RoboDK station: Double suction HAMK Robotics station MG400 Wood Sticks.rdk

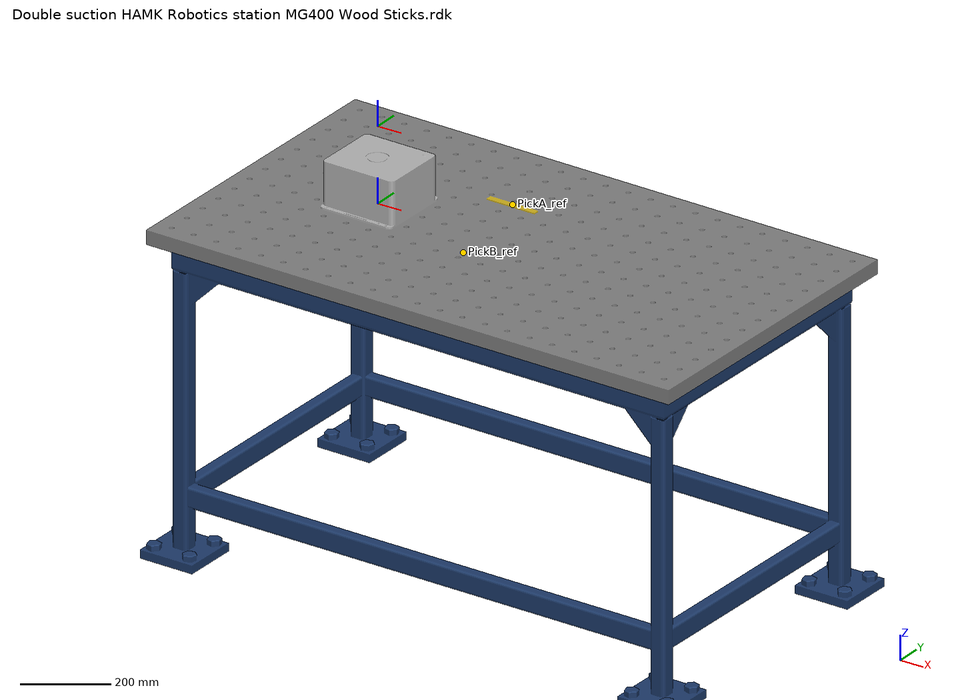
[picture v0: the station drawn from its stored meshes, robots at their saved joint values, targets as dots, program paths as lines]
Station Double suction HAMK Robotics Station MG400 Wood Sticks (saved by RoboDK 5.6.7). Poses are relative to the parent item; angles as X-Y-Z fixed-axis rotations.
Station parameters (name, value as stored): IO_1, 0, LIN64
  - frame Dobot MG400 Base at (0, 0, 0) mm
    - robot Dobot MG400: 4 axes, payload 0.5 kg, reach 393.5 mm, repeatability 0.2 mm, weight 4 kg
        joint limits [-160, -25, -25, -360] to [160, 85, 105, 360]; home [0, 0, 0, 0]; saved at [32.619, 68.287, 81.875, 32.609]
      - tool Suction Cup, TCP at (0, 0, 75.5) mm, size 42.6 x 40 x 76.8 mm
    - frame World at (0, 0, 0) mm
      - object Table 1400x800x800mm at (0, 0, 0) mm, size 1420 x 820 x 800 mm, geometry from Table-1400x800x800mm.sld
        - object HAMK logo at (360, 380, -115) mm, rotated rx 90 ry 0 rz 180 deg, size 301.4 x 100.9 x 9.4 mm, geometry from Fantastic Duup(2).stl
        - object white background at (360, 385.5, -110) mm, rotated rx 90 ry 0 rz 0 deg, size 480 x 184.8 x 2.4 mm, geometry from Fantastic Duup(3).stl
      - object Wood Stick at (250, 160, 0) mm, rotated rx 180 ry 0 rz 180 deg, size 128 x 15 x 3 mm, geometry from Wood Stick Biltema.stl
  - frame RefSuctionCup at (0, 0, 189) mm
    - target PickA_ref (Cartesian target) at (250, 160, -186) mm, rotated rx 180 ry 0 rz -179.99 deg; joints [32.619, 68.287, 81.875, 32.609] of Dobot MG400
    - target PickB_ref (Cartesian target) at (300, -100, -186) mm, rotated rx 180 ry 0 rz -179.99 deg; joints [-18.435, 69.533, 75.852, -18.445] of Dobot MG400
  - program StartPositions (2 instructions, listed below)

--- program StartPositions (robot Dobot MG400) ---
  Replace objects
  Show Wood Stick
